// TIA Portal project "Project6" (V17)

(* hardware
DEVICE "S7-1200 station_1"  S7-1200 Station
   slot 0: "Rack_0"  S7-1200 Rack  Rack  V1.0
   slot 1: "PLC_1"  CPU 1214C DC/DC/DC  6ES7 214-1AG40-0XB0  V4.5
*)

// ===== PLC "PLC_1"  CPU 1214C DC/DC/DC =====

VAR_GLOBAL   // PLC tag table "Default tag table"
   "S1" AT %I0.0 : Bool;
   "S2" AT %I0.1 : Bool;
   "LED1" AT %Q0.0 : Bool;
END_VAR

ORGANIZATION_BLOCK "Main"   // OB1, LAD, ProgramCycle
TITLE = "Main Program Sweep (Cycle)"
{ S7_Optimized_Access := 'TRUE' }
VERSION : 0.1
   VAR_INPUT
      Initial_Call : Bool;   // Initial call of this OB
      Remanence : Bool;   // =True, if remanent data are available
   END_VAR
BEGIN

REGION Network 1
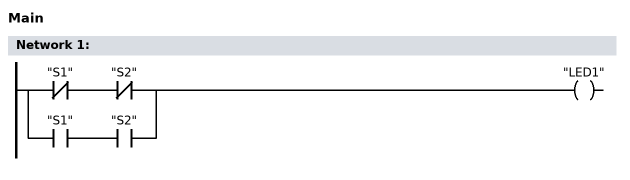
   RUNG wire#powerrail
      I_Contact( "S1" )
      I_Contact( "S2" )
      wire#w1
      Coil( "LED1" )
   END_RUNG
   RUNG wire#powerrail
      Contact( "S1" )
      Contact( "S2" )
   END_RUNG wire#w1
   // the same network as SCL:
   "LED1" := (NOT "S1" AND NOT "S2") OR ("S1" AND "S2");
END_REGION
END_ORGANIZATION_BLOCK